SUBAPPLICATION Uebung_012l_AX (* String Input und Speichern NVS *)
  (* Standard: 61499-2; Description: Copyright (c) 2026 Meisterschulen am Ostbahnhof This program and the accompanying materials are made available under the terms of the Eclipse Public License 2.0 which is available at https://www.eclipse.org/legal/epl-2.0/ SPDX-License-Identifier: EPL-2.0 *)
  (* Version 1.0, 2026-04-24, Franz Höpfinger, Meisterschulen am Ostbahnhof, AIS adapter variant of Uebung_012l *)
  PACKAGE Uebungen;
  IMPORT Uebungen::const::NVS::NVS_Keys::KEY_S1_STORE;
  IMPORT Uebungen::const::UT::DefaultPool::InputString_S1;
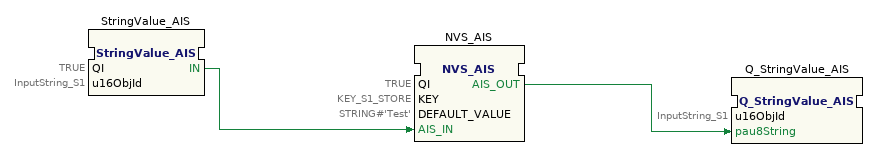
  FBS
    StringValue_AIS : isobus::UT::io::StringValue::StringValue_AIS(QI := TRUE, u16ObjId := InputString_S1);
    NVS_AIS : logiBUS::storage::esp32_nvs::NVS_AIS(QI := TRUE, KEY := KEY_S1_STORE, DEFAULT_VALUE := STRING#'Test');
    Q_StringValue_AIS : isobus::UT::Q::Q_StringValue_AIS(u16ObjId := InputString_S1);
  END_FBS
  ADAPTER_CONNECTIONS
    StringValue_AIS.IN TO NVS_AIS.AIS_IN;
    NVS_AIS.AIS_OUT TO Q_StringValue_AIS.pau8String;
  END_CONNECTIONS
END_SUBAPPLICATION
